                                FB_Bacnet.StartStopCommand_072.bEnWrite := TRUE;
                                FB_Bacnet.StartStopCommand_072.bVal := FALSE;
                            10: 
                                
                                FB_Bacnet.StartStopCommand_073.bEnWrite := TRUE;
                                FB_Bacnet.StartStopCommand_073.bVal := FALSE;
                            11: 
                                
                                FB_Bacnet.StartStopCommand_074.bEnWrite := TRUE;
                                FB_Bacnet.StartStopCommand_074.bVal := FALSE;
                            12: 
                                
                                FB_Bacnet.StartStopCommand_075.bEnWrite := TRUE;
                                FB_Bacnet.StartStopCommand_075.bVal := FALSE;
                            13: 
                                
                                FB_Bacnet.StartStopCommand_076.bEnWrite := TRUE;
                                FB_Bacnet.StartStopCommand_076.bVal := FALSE;
                            14: 
                                
                                FB_Bacnet.StartStopCommand_077.bEnWrite := TRUE;
                                FB_Bacnet.StartStopCommand_077.bVal := FALSE;
                            15: 
                                
                                FB_Bacnet.StartStopCommand_078.bEnWrite := TRUE;
                                FB_Bacnet.StartStopCommand_078.bVal := FALSE;
                            16: 
                                
                                FB_Bacnet.StartStopCommand_079.bEnWrite := TRUE;
                                FB_Bacnet.StartStopCommand_079.bVal := FALSE;
                            17: 
                                
                                FB_Bacnet.StartStopCommand_080.bEnWrite := TRUE;
                                FB_Bacnet.StartStopCommand_080.bVal := FALSE;
                            18: 
                                
                                FB_Bacnet.StartStopCommand_081.bEnWrite := TRUE;
                                FB_Bacnet.StartStopCommand_081.bVal := FALSE;
                            19: 
                                
                                FB_Bacnet.StartStopCommand_082.bEnWrite := TRUE;
                                FB_Bacnet.StartStopCommand_082.bVal := FALSE;
                            20: 
                                
                                FB_Bacnet.StartStopCommand_083.bEnWrite := TRUE;
                                FB_Bacnet.StartStopCommand_083.bVal := FALSE;
                            21: 
                                
                                FB_Bacnet.StartStopCommand_084.bEnWrite := TRUE;
                                FB_Bacnet.StartStopCommand_084.bVal := FALSE;
                            22: 
                                
                                FB_Bacnet.StartStopCommand_085.bEnWrite := TRUE;
                                FB_Bacnet.StartStopCommand_085.bVal := FALSE;
                            23: 
                                
                                FB_Bacnet.StartStopCommand_112.bEnWrite := TRUE;
                                FB_Bacnet.StartStopCommand_112.bVal := FALSE;
                            24: 
                                
                                FB_Bacnet.StartStopCommand_241.bEnWrite := TRUE;
                                FB_Bacnet.StartStopCommand_241.bVal := FALSE;
                            25: 
                                
                                FB_Bacnet.StartStopCommand_235.bEnWrite := TRUE;
                                FB_Bacnet.StartStopCommand_235.bVal := FALSE;
                        END_CASE
                    END_IF
                END_FOR
            END_IF
        END_IF
    END_IF
END_IF

END_FUNCTION_BLOCK

// ---- POUs/FB_Scheduler/FB_Scheduler_F52.TcPOU

      FUNCTION_BLOCK FB_Scheduler_F52
      VAR_INPUT
          currH : WORD;
          currM : WORD;
          currD : WORD;
      END_VAR
      VAR_IN_OUT
          FB_Bacnet : FB_BACnet_DAIKIN_MasterStation_III_No_10;
      END_VAR
      VAR
          i : INT;
          bUnitTriggered : BOOL := FALSE; // New flag to track execution
          prevMinute : WORD := 0;        // New variable to track the previous minute
      END_VAR
      VAR PERSISTENT
          //scheduler var
          bEnSchedF52_ : BOOL := FALSE;
          wSchedWDHourStartF52_ : WORD; 
          wSchedWDMinStartF52_ : WORD; 
          wSchedWEHourStartF52_ : WORD; 
          wSchedWEMinStartF52_ : WORD;
          wSchedWDHourEndF52_ : WORD;
          wSchedWDMinEndF52_ : WORD;
          wSchedWEHourEndF52_ : WORD;
          wSchedWEMinEndF52_ : WORD;
          //unit var
          bUnitF52_ : ARRAY [1..23] OF BOOL;
      END_VAR


        // Reset trigger flag at minute change or at the exact scheduled time
        IF currM <> prevMinute OR 
           (currH = wSchedWDHourStartF52_ AND currM = wSchedWDMinStartF52_) OR 
           (currH = wSchedWDHourEndF52_ AND currM = wSchedWDMinEndF52_) THEN
            bUnitTriggered := FALSE;
            prevMinute := currM;
        END_IF

        // Unit Schedule Enable
        IF bEnSchedF52_ THEN
            // Weekday schedule
            IF currD >= 1 AND currD <= 5 THEN
                IF (wSchedWDHourStartF52_ <> wSchedWDHourEndF52_ OR wSchedWDMinStartF52_ <> wSchedWDMinEndF52_) THEN
                    // Schedule Unit ON
                    IF wSchedWDHourStartF52_ = currH AND wSchedWDMinStartF52_ = currM AND NOT bUnitTriggered THEN
                        bUnitTriggered := TRUE;
                        FOR i := 1 TO 23 DO
                            //send command unit ON
                            IF bUnitF52_[i] = TRUE THEN 
                                CASE i OF
                                    1: 
                                        
                                        FB_Bacnet.StartStopCommand_128.bEnWrite := TRUE;
                                        FB_Bacnet.StartStopCommand_128.bVal := TRUE;
                                    2: 
                                        
                                        FB_Bacnet.StartStopCommand_129.bEnWrite := TRUE;
                                        FB_Bacnet.StartStopCommand_129.bVal := TRUE;
                                    3: 
                                        
                                        FB_Bacnet.StartStopCommand_130.bEnWrite := TRUE;
                                        FB_Bacnet.StartStopCommand_130.bVal := TRUE;
                                    4: 
                                        
                                        FB_Bacnet.StartStopCommand_131.bEnWrite := TRUE;
                                        FB_Bacnet.StartStopCommand_131.bVal := TRUE;
                                    5: 
                                        
                                        FB_Bacnet.StartStopCommand_132.bEnWrite := TRUE;
                                        FB_Bacnet.StartStopCommand_132.bVal := TRUE;
                                    6: 
                                        
                                        FB_Bacnet.StartStopCommand_133.bEnWrite := TRUE;
                                        FB_Bacnet.StartStopCommand_133.bVal := TRUE;
                                    7: 
                                        
                                        FB_Bacnet.StartStopCommand_134.bEnWrite := TRUE;
                                        FB_Bacnet.StartStopCommand_134.bVal := TRUE;
                                    8: 
                                        
                                        FB_Bacnet.StartStopCommand_135.bEnWrite := TRUE;
                                        FB_Bacnet.StartStopCommand_135.bVal := TRUE;
                                    9: 
                                        
                                        FB_Bacnet.StartStopCommand_136.bEnWrite := TRUE;
                                        FB_Bacnet.StartStopCommand_136.bVal := TRUE;
                                    10: 
                                        
                                        FB_Bacnet.StartStopCommand_137.bEnWrite := TRUE;
                                        FB_Bacnet.StartStopCommand_137.bVal := TRUE;
                                    11: 
                                        
                                        FB_Bacnet.StartStopCommand_138.bEnWrite := TRUE;
                                        FB_Bacnet.StartStopCommand_138.bVal := TRUE;
                                    12: 
                                        
                                        FB_Bacnet.StartStopCommand_139.bEnWrite := TRUE;
                                        FB_Bacnet.StartStopCommand_139.bVal := TRUE;
                                    13: 
                                        
                                        FB_Bacnet.StartStopCommand_140.bEnWrite := TRUE;
                                        FB_Bacnet.StartStopCommand_140.bVal := TRUE;
                                    14: 
                                        
                                        FB_Bacnet.StartStopCommand_141.bEnWrite := TRUE;
                                        FB_Bacnet.StartStopCommand_141.bVal := TRUE;
                                    15: 
                                        
                                        FB_Bacnet.StartStopCommand_142.bEnWrite := TRUE;
                                        FB_Bacnet.StartStopCommand_142.bVal := TRUE;
                                    16: 
                                        
                                        FB_Bacnet.StartStopCommand_143.bEnWrite := TRUE;
                                        FB_Bacnet.StartStopCommand_143.bVal := TRUE;
                                    17: 
                                        
                                        FB_Bacnet.StartStopCommand_144.bEnWrite := TRUE;
                                        FB_Bacnet.StartStopCommand_144.bVal := TRUE;
                                    18: 
                                        
                                        FB_Bacnet.StartStopCommand_145.bEnWrite := TRUE;
                                        FB_Bacnet.StartStopCommand_145.bVal := TRUE;
                                    19: 
                                        
                                        FB_Bacnet.StartStopCommand_146.bEnWrite := TRUE;
                                        FB_Bacnet.StartStopCommand_146.bVal := TRUE;
                                    20: 
                                        
                                        FB_Bacnet.StartStopCommand_147.bEnWrite := TRUE;
                                        FB_Bacnet.StartStopCommand_147.bVal := TRUE;
                                    21: 
                                        
                                        FB_Bacnet.StartStopCommand_148.bEnWrite := TRUE;
                                        FB_Bacnet.StartStopCommand_148.bVal := TRUE;
                                    22: 
                                        
                                        FB_Bacnet.StartStopCommand_149.bEnWrite := TRUE;
                                        FB_Bacnet.StartStopCommand_149.bVal := TRUE;
                                    23: 
                                        
                                        FB_Bacnet.StartStopCommand_236.bEnWrite := TRUE;
                                        FB_Bacnet.StartStopCommand_236.bVal := TRUE;
                                END_CASE
                            END_IF
                        END_FOR
                    END_IF
                    // Schedule Unit OFF
                    IF wSchedWDHourEndF52_ = currH AND wSchedWDMinEndF52_ = currM AND NOT bUnitTriggered THEN
                        bUnitTriggered := TRUE;
                        FOR i := 1 TO 23 DO
                            //send command unit OFF
                            IF bUnitF52_[i] = TRUE THEN 
                                CASE i OF
                                    1: 
                                        
                                        FB_Bacnet.StartStopCommand_128.bEnWrite := TRUE;
                                        FB_Bacnet.StartStopCommand_128.bVal := FALSE;
                                    2: 
                                        
                                        FB_Bacnet.StartStopCommand_129.bEnWrite := TRUE;
                                        FB_Bacnet.StartStopCommand_129.bVal := FALSE;
                                    3: 
                                        
                                        FB_Bacnet.StartStopCommand_130.bEnWrite := TRUE;
                                        FB_Bacnet.StartStopCommand_130.bVal := FALSE;
                                    4: 
                                        
                                        FB_Bacnet.StartStopCommand_131.bEnWrite := TRUE;
                                        FB_Bacnet.StartStopCommand_131.bVal := FALSE;
                                    5: 
                                        
                                        FB_Bacnet.StartStopCommand_132.bEnWrite := TRUE;
                                        FB_Bacnet.StartStopCommand_132.bVal := FALSE;
                                    6: 
                                        
                                        FB_Bacnet.StartStopCommand_133.bEnWrite := TRUE;
                                        FB_Bacnet.StartStopCommand_133.bVal := FALSE;
                                    7: 
                                        
                                        FB_Bacnet.StartStopCommand_134.bEnWrite := TRUE;
                                        FB_Bacnet.StartStopCommand_134.bVal := FALSE;
                                    8: 
                                        
                                        FB_Bacnet.StartStopCommand_135.bEnWrite := TRUE;
                                        FB_Bacnet.StartStopCommand_135.bVal := FALSE;
                                    9: 
                                        
                                        FB_Bacnet.StartStopCommand_136.bEnWrite := TRUE;
                                        FB_Bacnet.StartStopCommand_136.bVal := FALSE;
                                    10: 
                                        
                                        FB_Bacnet.StartStopCommand_137.bEnWrite := TRUE;
                                        FB_Bacnet.StartStopCommand_137.bVal := FALSE;
                                    11: 
                                        
                                        FB_Bacnet.StartStopCommand_138.bEnWrite := TRUE;
                                        FB_Bacnet.StartStopCommand_138.bVal := FALSE;
                                    12: 
                                        
                                        FB_Bacnet.StartStopCommand_139.bEnWrite := TRUE;
                                        FB_Bacnet.StartStopCommand_139.bVal := FALSE;
                                    13: 
                                        
                                        FB_Bacnet.StartStopCommand_140.bEnWrite := TRUE;
                                        FB_Bacnet.StartStopCommand_140.bVal := FALSE;
                                    14: 
                                        
                                        FB_Bacnet.StartStopCommand_141.bEnWrite := TRUE;
                                        FB_Bacnet.StartStopCommand_141.bVal := FALSE;
                                    15: 
                                        
                                        FB_Bacnet.StartStopCommand_142.bEnWrite := TRUE;
                                        FB_Bacnet.StartStopCommand_142.bVal := FALSE;
                                    16: 
                                        
                                        FB_Bacnet.StartStopCommand_143.bEnWrite := TRUE;
                                        FB_Bacnet.StartStopCommand_143.bVal := FALSE;
                                    17: 
                                        
                                        FB_Bacnet.StartStopCommand_144.bEnWrite := TRUE;
                                        FB_Bacnet.StartStopCommand_144.bVal := FALSE;
                                    18: 
                                        
                                        FB_Bacnet.StartStopCommand_145.bEnWrite := TRUE;
                                        FB_Bacnet.StartStopCommand_145.bVal := FALSE;
                                    19: 
                                        
                                        FB_Bacnet.StartStopCommand_146.bEnWrite := TRUE;
                                        FB_Bacnet.StartStopCommand_146.bVal := FALSE;
                                    20: 
                                        
                                        FB_Bacnet.StartStopCommand_147.bEnWrite := TRUE;
                                        FB_Bacnet.StartStopCommand_147.bVal := FALSE;
                                    21: 
                                        
                                        FB_Bacnet.StartStopCommand_148.bEnWrite := TRUE;
                                        FB_Bacnet.StartStopCommand_148.bVal := FALSE;
                                    22: 
                                        
                                        FB_Bacnet.StartStopCommand_149.bEnWrite := TRUE;
                                        FB_Bacnet.StartStopCommand_149.bVal := FALSE;
                                    23: 
                                        
                                        FB_Bacnet.StartStopCommand_236.bEnWrite := TRUE;
                                        FB_Bacnet.StartStopCommand_236.bVal := FALSE;
                                END_CASE
                            END_IF
                        END_FOR
                    END_IF
                END_IF
            END_IF

            // Weekend schedule
            IF currD = 0 OR currD = 6 THEN
                IF (wSchedWEHourStartF52_ <> wSchedWEHourEndF52_ OR wSchedWEMinStartF52_ <> wSchedWEMinEndF52_) THEN
                    // Schedule Unit ON
                    IF wSchedWEHourStartF52_ = currH AND wSchedWEMinStartF52_ = currM AND NOT bUnitTriggered THEN
                        bUnitTriggered := TRUE;
                        FOR i := 1 TO 23 DO
                            //send command unit ON
                            IF bUnitF52_[i] = TRUE THEN 
                                CASE i OF
                                    1: 
                                        
                                        FB_Bacnet.StartStopCommand_128.bEnWrite := TRUE;
                                        FB_Bacnet.StartStopCommand_128.bVal := TRUE;
                                    2: 
                                        
                                        FB_Bacnet.StartStopCommand_129.bEnWrite := TRUE;
                                        FB_Bacnet.StartStopCommand_129.bVal := TRUE;
                                    3: 
                                        
                                        FB_Bacnet.StartStopCommand_130.bEnWrite := TRUE;
                                        FB_Bacnet.StartStopCommand_130.bVal := TRUE;
                                    4: 
                                        
                                        FB_Bacnet.StartStopCommand_131.bEnWrite := TRUE;
                                        FB_Bacnet.StartStopCommand_131.bVal := TRUE;
                                    5: 
                                        
                                        FB_Bacnet.StartStopCommand_132.bEnWrite := TRUE;
                                        FB_Bacnet.StartStopCommand_132.bVal := TRUE;
                                    6: 
                                        
                                        FB_Bacnet.StartStopCommand_133.bEnWrite := TRUE;
                                        FB_Bacnet.StartStopCommand_133.bVal := TRUE;
                                    7: 
                                        
                                        FB_Bacnet.StartStopCommand_134.bEnWrite := TRUE;
                                        FB_Bacnet.StartStopCommand_134.bVal := TRUE;
                                    8: 
                                        
                                        FB_Bacnet.StartStopCommand_135.bEnWrite := TRUE;
                                        FB_Bacnet.StartStopCommand_135.bVal := TRUE;
                                    9: 
                                        
                                        FB_Bacnet.StartStopCommand_136.bEnWrite := TRUE;
                                        FB_Bacnet.StartStopCommand_136.bVal := TRUE;
                                    10: 
                                        
                                        FB_Bacnet.StartStopCommand_137.bEnWrite := TRUE;
                                        FB_Bacnet.StartStopCommand_137.bVal := TRUE;
                                    11: 
                                        
                                        FB_Bacnet.StartStopCommand_138.bEnWrite := TRUE;
                                        FB_Bacnet.StartStopCommand_138.bVal := TRUE;
                                    12: 
                                        
                                        FB_Bacnet.StartStopCommand_139.bEnWrite := TRUE;
                                        FB_Bacnet.StartStopCommand_139.bVal := TRUE;
                                    13: 
                                        
                                        FB_Bacnet.StartStopCommand_140.bEnWrite := TRUE;
                                        FB_Bacnet.StartStopCommand_140.bVal := TRUE;
                                    14: 
                                        
                                        FB_Bacnet.StartStopCommand_141.bEnWrite := TRUE;
                                        FB_Bacnet.StartStopCommand_141.bVal := TRUE;
                                    15: 
                                        
                                        FB_Bacnet.StartStopCommand_142.bEnWrite := TRUE;
                                        FB_Bacnet.StartStopCommand_142.bVal := TRUE;
                                    16: 
                                        
                                        FB_Bacnet.StartStopCommand_143.bEnWrite := TRUE;
                                        FB_Bacnet.StartStopCommand_143.bVal := TRUE;
                                    17: 
                                        
                                        FB_Bacnet.StartStopCommand_144.bEnWrite := TRUE;
                                        FB_Bacnet.StartStopCommand_144.bVal := TRUE;
                                    18: 
                                        
                                        FB_Bacnet.StartStopCommand_145.bEnWrite := TRUE;
                                        FB_Bacnet.StartStopCommand_145.bVal := TRUE;
                                    19: 
                                        
                                        FB_Bacnet.StartStopCommand_146.bEnWrite := TRUE;
                                        FB_Bacnet.StartStopCommand_146.bVal := TRUE;
                                    20: 
                                        
                                        FB_Bacnet.StartStopCommand_147.bEnWrite := TRUE;
                                        FB_Bacnet.StartStopCommand_147.bVal := TRUE;
                                    21: 
                                        
                                        FB_Bacnet.StartStopCommand_148.bEnWrite := TRUE;
                                        FB_Bacnet.StartStopCommand_148.bVal := TRUE;
                                    22: 
                                        
                                        FB_Bacnet.StartStopCommand_149.bEnWrite := TRUE;
                                        FB_Bacnet.StartStopCommand_149.bVal := TRUE;
                                    23: 
                                        
                                        FB_Bacnet.StartStopCommand_236.bEnWrite := TRUE;
                                        FB_Bacnet.StartStopCommand_236.bVal := TRUE;
                                END_CASE
                            END_IF
                        END_FOR
                    END_IF
                    // Schedule Unit OFF
                    IF wSchedWEHourEndF52_ = currH AND wSchedWEMinEndF52_ = currM AND NOT bUnitTriggered THEN
                        bUnitTriggered := TRUE;
                        FOR i := 1 TO 23 DO
                            //send command unit OFF
                            IF bUnitF52_[i] = TRUE THEN 
                                CASE i OF
                                    1: 
                                        
                                        FB_Bacnet.StartStopCommand_128.bEnWrite := TRUE;
                                        FB_Bacnet.StartStopCommand_128.bVal := FALSE;
                                    2: 
                                        
                                        FB_Bacnet.StartStopCommand_129.bEnWrite := TRUE;
                                        FB_Bacnet.StartStopCommand_129.bVal := FALSE;
                                    3: 
                                        
                                        FB_Bacnet.StartStopCommand_130.bEnWrite := TRUE;
                                        FB_Bacnet.StartStopCommand_130.bVal := FALSE;
                                    4: 
                                        
                                        FB_Bacnet.StartStopCommand_131.bEnWrite := TRUE;
                                        FB_Bacnet.StartStopCommand_131.bVal := FALSE;
                                    5: 
                                        
                                        FB_Bacnet.StartStopCommand_132.bEnWrite := TRUE;
                                        FB_Bacnet.StartStopCommand_132.bVal := FALSE;
                                    6: 
                                        
                                        FB_Bacnet.StartStopCommand_133.bEnWrite := TRUE;
                                        FB_Bacnet.StartStopCommand_133.bVal := FALSE;
                                    7: 
                                        
                                        FB_Bacnet.StartStopCommand_134.bEnWrite := TRUE;
                                        FB_Bacnet.StartStopCommand_134.bVal := FALSE;
                                    8: 
                                        
                                        FB_Bacnet.StartStopCommand_135.bEnWrite := TRUE;
                                        FB_Bacnet.StartStopCommand_135.bVal := FALSE;
                                    9: 
                                        
                                        FB_Bacnet.StartStopCommand_136.bEnWrite := TRUE;
                                        FB_Bacnet.StartStopCommand_136.bVal := FALSE;
                                    10: 
                                        
                                        FB_Bacnet.StartStopCommand_137.bEnWrite := TRUE;
                                        FB_Bacnet.StartStopCommand_137.bVal := FALSE;
                                    11: 
                                        
                                        FB_Bacnet.StartStopCommand_138.bEnWrite := TRUE;
                                        FB_Bacnet.StartStopCommand_138.bVal := FALSE;
                                    12: 
                                        
                                        FB_Bacnet.StartStopCommand_139.bEnWrite := TRUE;
                                        FB_Bacnet.StartStopCommand_139.bVal := FALSE;
                                    13: 
                                        
                                        FB_Bacnet.StartStopCommand_140.bEnWrite := TRUE;
                                        FB_Bacnet.StartStopCommand_140.bVal := FALSE;
                                    14: 
                                        
                                        FB_Bacnet.StartStopCommand_141.bEnWrite := TRUE;
                                        FB_Bacnet.StartStopCommand_141.bVal := FALSE;
                                    15: 
                                        
                                        FB_Bacnet.StartStopCommand_142.bEnWrite := TRUE;
                                        FB_Bacnet.StartStopCommand_142.bVal := FALSE;
                                    16: 
                                        
                                        FB_Bacnet.StartStopCommand_143.bEnWrite := TRUE;
                                        FB_Bacnet.StartStopCommand_143.bVal := FALSE;
                                    17: 
                                        
                                        FB_Bacnet.StartStopCommand_144.bEnWrite := TRUE;
                                        FB_Bacnet.StartStopCommand_144.bVal := FALSE;
                                    18: 
                                        
                                        FB_Bacnet.StartStopCommand_145.bEnWrite := TRUE;
                                        FB_Bacnet.StartStopCommand_145.bVal := FALSE;
                                    19: 
                                        
                                        FB_Bacnet.StartStopCommand_146.bEnWrite := TRUE;
                                        FB_Bacnet.StartStopCommand_146.bVal := FALSE;
                                    20: 
                                        
                                        FB_Bacnet.StartStopCommand_147.bEnWrite := TRUE;
                                        FB_Bacnet.StartStopCommand_147.bVal := FALSE;
                                    21: 
                                        
                                        FB_Bacnet.StartStopCommand_148.bEnWrite := TRUE;
                                        FB_Bacnet.StartStopCommand_148.bVal := FALSE;
                                    22: 
                                        
                                        FB_Bacnet.StartStopCommand_149.bEnWrite := TRUE;
                                        FB_Bacnet.StartStopCommand_149.bVal := FALSE;
                                    23: 
                                        
                                        FB_Bacnet.StartStopCommand_236.bEnWrite := TRUE;
                                        FB_Bacnet.StartStopCommand_236.bVal := FALSE;
                                END_CASE
                            END_IF
                        END_FOR
                    END_IF
                END_IF
            END_IF
        END_IF

END_FUNCTION_BLOCK

// ---- POUs/FB_Scheduler/FB_Scheduler_F53.TcPOU

    FUNCTION_BLOCK FB_Scheduler_F53
      VAR_INPUT
          currH : WORD;
          currM : WORD;
          currD : WORD;
      END_VAR
      VAR_IN_OUT
          FB_Bacnet : FB_BACnet_DAIKIN_MasterStation_III_No_10;
      END_VAR
      VAR
          i : INT;
          bUnitTriggered : BOOL := FALSE; // New flag to track execution
          prevMinute : WORD := 0;        // New variable to track the previous minute
      END_VAR
      VAR PERSISTENT
          //scheduler var
          bEnSchedF53_ : BOOL := FALSE;
          wSchedWDHourStartF53_ : WORD; 
          wSchedWDMinStartF53_ : WORD; 
          wSchedWEHourStartF53_ : WORD; 
          wSchedWEMinStartF53_ : WORD;
          wSchedWDHourEndF53_ : WORD;
          wSchedWDMinEndF53_ : WORD;
          wSchedWEHourEndF53_ : WORD;
          wSchedWEMinEndF53_ : WORD;
          //unit var
          bUnitF53_ : ARRAY [1..25] OF BOOL;
      END_VAR


// Reset trigger flag at minute change or at the exact scheduled time
IF currM <> prevMinute OR 
   (currH = wSchedWDHourStartF53_ AND currM = wSchedWDMinStartF53_) OR 
   (currH = wSchedWDHourEndF53_ AND currM = wSchedWDMinEndF53_) THEN
    bUnitTriggered := FALSE;
    prevMinute := currM;
END_IF

// Unit Schedule Enable
IF bEnSchedF53_ THEN
    // Weekday schedule
    IF currD >= 1 AND currD <= 5 THEN
        IF (wSchedWDHourStartF53_ <> wSchedWDHourEndF53_ OR wSchedWDMinStartF53_ <> wSchedWDMinEndF53_) THEN
            // Schedule Unit ON
            IF wSchedWDHourStartF53_ = currH AND wSchedWDMinStartF53_ = currM AND NOT bUnitTriggered THEN
                bUnitTriggered := TRUE;
                FOR i := 1 TO 25 DO
                    //send command unit ON
                    IF bUnitF53_[i] = TRUE THEN 
                        CASE i OF
                            1: 
                                FB_Bacnet.StartStopCommand_192.bEnWrite := TRUE;
                                FB_Bacnet.StartStopCommand_192.bVal := TRUE;
                            2: 
                                FB_Bacnet.StartStopCommand_193.bEnWrite := TRUE;
                                FB_Bacnet.StartStopCommand_193.bVal := TRUE;
                            3: 
                                FB_Bacnet.StartStopCommand_194.bEnWrite := TRUE;
                                FB_Bacnet.StartStopCommand_194.bVal := TRUE;
                            4: 
                                FB_Bacnet.StartStopCommand_195.bEnWrite := TRUE;
                                FB_Bacnet.StartStopCommand_195.bVal := TRUE;
                            5: 
                                FB_Bacnet.StartStopCommand_196.bEnWrite := TRUE;
                                FB_Bacnet.StartStopCommand_196.bVal := TRUE;
                            6: 
                                FB_Bacnet.StartStopCommand_197.bEnWrite := TRUE;
                                FB_Bacnet.StartStopCommand_197.bVal := TRUE;
                            7: 
                                FB_Bacnet.StartStopCommand_198.bEnWrite := TRUE;
                                FB_Bacnet.StartStopCommand_198.bVal := TRUE;
                            8: 
                                FB_Bacnet.StartStopCommand_199.bEnWrite := TRUE;
                                FB_Bacnet.StartStopCommand_199.bVal := TRUE;
                            9: 
                                //FB_Bacnet.StartStopCommand_200.bEnWrite := TRUE;
                                //FB_Bacnet.StartStopCommand_200.bVal := TRUE;
                            10: 
                                FB_Bacnet.StartStopCommand_201.bEnWrite := TRUE;
                                FB_Bacnet.StartStopCommand_201.bVal := TRUE;
                            11: 
                                FB_Bacnet.StartStopCommand_202.bEnWrite := TRUE;
                                FB_Bacnet.StartStopCommand_202.bVal := TRUE;
                            12: 
                                FB_Bacnet.StartStopCommand_203.bEnWrite := TRUE;
                                FB_Bacnet.StartStopCommand_203.bVal := TRUE;
                            13: 
                                FB_Bacnet.StartStopCommand_204.bEnWrite := TRUE;
                                FB_Bacnet.StartStopCommand_204.bVal := TRUE;
                            14: 
                                FB_Bacnet.StartStopCommand_205.bEnWrite := TRUE;
                                FB_Bacnet.StartStopCommand_205.bVal := TRUE;
                            15: 
                                FB_Bacnet.StartStopCommand_206.bEnWrite := TRUE;
                                FB_Bacnet.StartStopCommand_206.bVal := TRUE;
                            16: 
                                FB_Bacnet.StartStopCommand_207.bEnWrite := TRUE;
                                FB_Bacnet.StartStopCommand_207.bVal := TRUE;
                            17: 
                                FB_Bacnet.StartStopCommand_208.bEnWrite := TRUE;
                                FB_Bacnet.StartStopCommand_208.bVal := TRUE;
                            18: 
                                FB_Bacnet.StartStopCommand_209.bEnWrite := TRUE;
                                FB_Bacnet.StartStopCommand_209.bVal := TRUE;
                            19: 
                                FB_Bacnet.StartStopCommand_210.bEnWrite := TRUE;
                                FB_Bacnet.StartStopCommand_210.bVal := TRUE;
                            20: 
                                FB_Bacnet.StartStopCommand_211.bEnWrite := TRUE;
                                FB_Bacnet.StartStopCommand_211.bVal := TRUE;
                            21: 
                                FB_Bacnet.StartStopCommand_212.bEnWrite := TRUE;
                                FB_Bacnet.StartStopCommand_212.bVal := TRUE;
                            22: 
                                FB_Bacnet.StartStopCommand_213.bEnWrite := TRUE;
                                FB_Bacnet.StartStopCommand_213.bVal := TRUE;
                            23: 
                                FB_Bacnet.StartStopCommand_242.bEnWrite := TRUE;
                                FB_Bacnet.StartStopCommand_242.bVal := TRUE;
                            24: 
                                FB_Bacnet.StartStopCommand_243.bEnWrite := TRUE;
                                FB_Bacnet.StartStopCommand_243.bVal := TRUE;
                            25: 
                                FB_Bacnet.StartStopCommand_237.bEnWrite := TRUE;
                                FB_Bacnet.StartStopCommand_237.bVal := TRUE;
                        END_CASE
                    END_IF
                END_FOR
            END_IF
            // Schedule Unit OFF
            IF wSchedWDHourEndF53_ = currH AND wSchedWDMinEndF53_ = currM AND NOT bUnitTriggered THEN
                bUnitTriggered := TRUE;
                FOR i := 1 TO 25 DO
                    //send command unit OFF
                    IF bUnitF53_[i] = TRUE THEN 
                        CASE i OF
                            1: 
                                FB_Bacnet.StartStopCommand_192.bEnWrite := TRUE;
                                FB_Bacnet.StartStopCommand_192.bVal := FALSE;
                            2: 
                                FB_Bacnet.StartStopCommand_193.bEnWrite := TRUE;
                                FB_Bacnet.StartStopCommand_193.bVal := FALSE;
                            3: 
                                FB_Bacnet.StartStopCommand_194.bEnWrite := TRUE;
                                FB_Bacnet.StartStopCommand_194.bVal := FALSE;
                            4: 
                                FB_Bacnet.StartStopCommand_195.bEnWrite := TRUE;
                                FB_Bacnet.StartStopCommand_195.bVal := FALSE;
                            5: 
                                FB_Bacnet.StartStopCommand_196.bEnWrite := TRUE;
                                FB_Bacnet.StartStopCommand_196.bVal := FALSE;
                            6: 
                                FB_Bacnet.StartStopCommand_197.bEnWrite := TRUE;
                                FB_Bacnet.StartStopCommand_197.bVal := FALSE;
                            7: 
                                FB_Bacnet.StartStopCommand_198.bEnWrite := TRUE;
                                FB_Bacnet.StartStopCommand_198.bVal := FALSE;
                            8: 
                                FB_Bacnet.StartStopCommand_199.bEnWrite := TRUE;
                                FB_Bacnet.StartStopCommand_199.bVal := FALSE;
                            9: 
                                //FB_Bacnet.StartStopCommand_200.bEnWrite := TRUE;
                                //FB_Bacnet.StartStopCommand_200.bVal := FALSE;
                            10: 
                                FB_Bacnet.StartStopCommand_201.bEnWrite := TRUE;
                                FB_Bacnet.StartStopCommand_201.bVal := FALSE;
                            11: 
                                FB_Bacnet.StartStopCommand_202.bEnWrite := TRUE;
                                FB_Bacnet.StartStopCommand_202.bVal := FALSE;
                            12: 
                                FB_Bacnet.StartStopCommand_203.bEnWrite := TRUE;
                                FB_Bacnet.StartStopCommand_203.bVal := FALSE;
                            13: 
                                FB_Bacnet.StartStopCommand_204.bEnWrite := TRUE;
                                FB_Bacnet.StartStopCommand_204.bVal := FALSE;
                            14: 
                                FB_Bacnet.StartStopCommand_205.bEnWrite := TRUE;
                                FB_Bacnet.StartStopCommand_205.bVal := FALSE;
                            15: 
                                FB_Bacnet.StartStopCommand_206.bEnWrite := TRUE;
                                FB_Bacnet.StartStopCommand_206.bVal := FALSE;
                            16: 
                                FB_Bacnet.StartStopCommand_207.bEnWrite := TRUE;
                                FB_Bacnet.StartStopCommand_207.bVal := FALSE;
                            17: 
                                FB_Bacnet.StartStopCommand_208.bEnWrite := TRUE;
                                FB_Bacnet.StartStopCommand_208.bVal := FALSE;
                            18: 
                                FB_Bacnet.StartStopCommand_209.bEnWrite := TRUE;
                                FB_Bacnet.StartStopCommand_209.bVal := FALSE;
                            19: 
                                FB_Bacnet.StartStopCommand_210.bEnWrite := TRUE;
                                FB_Bacnet.StartStopCommand_210.bVal := FALSE;
                            20: 
                                FB_Bacnet.StartStopCommand_211.bEnWrite := TRUE;
                                FB_Bacnet.StartStopCommand_211.bVal := FALSE;
                            21: 
                                FB_Bacnet.StartStopCommand_212.bEnWrite := TRUE;
                                FB_Bacnet.StartStopCommand_212.bVal := FALSE;
                            22: 
                                FB_Bacnet.StartStopCommand_213.bEnWrite := TRUE;
                                FB_Bacnet.StartStopCommand_213.bVal := FALSE;
                            23: 
                                FB_Bacnet.StartStopCommand_242.bEnWrite := TRUE;
                                FB_Bacnet.StartStopCommand_242.bVal := FALSE;
                            24: 
                                FB_Bacnet.StartStopCommand_243.bEnWrite := TRUE;
                                FB_Bacnet.StartStopCommand_243.bVal := FALSE;
                            25: 
                                FB_Bacnet.StartStopCommand_237.bEnWrite := TRUE;
                                FB_Bacnet.StartStopCommand_237.bVal := FALSE;
                        END_CASE
                    END_IF
                END_FOR
            END_IF
        END_IF
    END_IF

    // Weekend schedule
    IF currD = 0 OR currD = 6 THEN
        IF (wSchedWEHourStartF53_ <> wSchedWEHourEndF53_ OR wSchedWEMinStartF53_ <> wSchedWEMinEndF53_) THEN
            // Schedule Unit ON
            IF wSchedWEHourStartF53_ = currH AND wSchedWEMinStartF53_ = currM AND NOT bUnitTriggered THEN
                bUnitTriggered := TRUE;
                FOR i := 1 TO 25 DO
                    //send command unit ON
                    IF bUnitF53_[i] = TRUE THEN 
                        CASE i OF
                            1: 
                                FB_Bacnet.StartStopCommand_192.bEnWrite := TRUE;
                                FB_Bacnet.StartStopCommand_192.bVal := TRUE;
                            2: 
                                FB_Bacnet.StartStopCommand_193.bEnWrite := TRUE;
                                FB_Bacnet.StartStopCommand_193.bVal := TRUE;
                            3: 
                                FB_Bacnet.StartStopCommand_194.bEnWrite := TRUE;
                                FB_Bacnet.StartStopCommand_194.bVal := TRUE;
                            4: 
                                FB_Bacnet.StartStopCommand_195.bEnWrite := TRUE;
                                FB_Bacnet.StartStopCommand_195.bVal := TRUE;
                            5: 
                                FB_Bacnet.StartStopCommand_196.bEnWrite := TRUE;
                                FB_Bacnet.StartStopCommand_196.bVal := TRUE;
                            6: 
                                FB_Bacnet.StartStopCommand_197.bEnWrite := TRUE;
                                FB_Bacnet.StartStopCommand_197.bVal := TRUE;
                            7: 
                                FB_Bacnet.StartStopCommand_198.bEnWrite := TRUE;
                                FB_Bacnet.StartStopCommand_198.bVal := TRUE;
                            8: 
                                FB_Bacnet.StartStopCommand_199.bEnWrite := TRUE;
                                FB_Bacnet.StartStopCommand_199.bVal := TRUE;
                            9: 
                                //FB_Bacnet.StartStopCommand_200.bEnWrite := TRUE;
                                //FB_Bacnet.StartStopCommand_200.bVal := TRUE;
                            10: 
                                FB_Bacnet.StartStopCommand_201.bEnWrite := TRUE;
                                FB_Bacnet.StartStopCommand_201.bVal := TRUE;
                            11: 
                                FB_Bacnet.StartStopCommand_202.bEnWrite := TRUE;
                                FB_Bacnet.StartStopCommand_202.bVal := TRUE;
                            12: 
                                FB_Bacnet.StartStopCommand_203.bEnWrite := TRUE;
                                FB_Bacnet.StartStopCommand_203.bVal := TRUE;
                            13: 
                                FB_Bacnet.StartStopCommand_204.bEnWrite := TRUE;
                                FB_Bacnet.StartStopCommand_204.bVal := TRUE;
                            14: 
                                FB_Bacnet.StartStopCommand_205.bEnWrite := TRUE;
                                FB_Bacnet.StartStopCommand_205.bVal := TRUE;
                            15: 
                                FB_Bacnet.StartStopCommand_206.bEnWrite := TRUE;
                                FB_Bacnet.StartStopCommand_206.bVal := TRUE;
                            16: 
                                FB_Bacnet.StartStopCommand_207.bEnWrite := TRUE;
                                FB_Bacnet.StartStopCommand_207.bVal := TRUE;
                            17: 
                                FB_Bacnet.StartStopCommand_208.bEnWrite := TRUE;
                                FB_Bacnet.StartStopCommand_208.bVal := TRUE;
                            18: 
                                FB_Bacnet.StartStopCommand_209.bEnWrite := TRUE;
                                FB_Bacnet.StartStopCommand_209.bVal := TRUE;
                            19: 
                                FB_Bacnet.StartStopCommand_210.bEnWrite := TRUE;
                                FB_Bacnet.StartStopCommand_210.bVal := TRUE;
                            20: 
                                FB_Bacnet.StartStopCommand_211.bEnWrite := TRUE;
                                FB_Bacnet.StartStopCommand_211.bVal := TRUE;
                            21: 
                                FB_Bacnet.StartStopCommand_212.bEnWrite := TRUE;
                                FB_Bacnet.StartStopCommand_212.bVal := TRUE;
                            22: 
                                FB_Bacnet.StartStopCommand_213.bEnWrite := TRUE;
                                FB_Bacnet.StartStopCommand_213.bVal := TRUE;
                            23: 
                                FB_Bacnet.StartStopCommand_242.bEnWrite := TRUE;
                                FB_Bacnet.StartStopCommand_242.bVal := TRUE;
                            24: 
                                FB_Bacnet.StartStopCommand_243.bEnWrite := TRUE;
                                FB_Bacnet.StartStopCommand_243.bVal := TRUE;
                            25: 
                                FB_Bacnet.StartStopCommand_237.bEnWrite := TRUE;
                                FB_Bacnet.StartStopCommand_237.bVal := TRUE;
                        END_CASE
                    END_IF
                END_FOR        
            END_IF
            // Schedule Unit OFF
            IF wSchedWEHourEndF53_ = currH AND wSchedWEMinEndF53_ = currM AND NOT bUnitTriggered THEN
                bUnitTriggered := TRUE;
                FOR i := 1 TO 25 DO
                    //send command unit OFF
                    IF bUnitF53_[i] = TRUE THEN 
                        CASE i OF
                            1: 
                                FB_Bacnet.StartStopCommand_192.bEnWrite := TRUE;
                                FB_Bacnet.StartStopCommand_192.bVal := FALSE;
                            2: 
                                FB_Bacnet.StartStopCommand_193.bEnWrite := TRUE;
                                FB_Bacnet.StartStopCommand_193.bVal := FALSE;
                            3: 
                                FB_Bacnet.StartStopCommand_194.bEnWrite := TRUE;
                                FB_Bacnet.StartStopCommand_194.bVal := FALSE;
                            4: 
                                FB_Bacnet.StartStopCommand_195.bEnWrite := TRUE;
                                FB_Bacnet.StartStopCommand_195.bVal := FALSE;
                            5: 
                                FB_Bacnet.StartStopCommand_196.bEnWrite := TRUE;
                                FB_Bacnet.StartStopCommand_196.bVal := FALSE;
                            6: 
                                FB_Bacnet.StartStopCommand_197.bEnWrite := TRUE;
                                FB_Bacnet.StartStopCommand_197.bVal := FALSE;
                            7: 
                                FB_Bacnet.StartStopCommand_198.bEnWrite := TRUE;
                                FB_Bacnet.StartStopCommand_198.bVal := FALSE;
                            8: 
                                FB_Bacnet.StartStopCommand_199.bEnWrite := TRUE;
                                FB_Bacnet.StartStopCommand_199.bVal := FALSE;
                            9: 
                                //FB_Bacnet.StartStopCommand_200.bEnWrite := TRUE;
                                //FB_Bacnet.StartStopCommand_200.bVal := FALSE;
                            10: 
                                FB_Bacnet.StartStopCommand_201.bEnWrite := TRUE;
                                FB_Bacnet.StartStopCommand_201.bVal := FALSE;
                            11: 
                                FB_Bacnet.StartStopCommand_202.bEnWrite := TRUE;
                                FB_Bacnet.StartStopCommand_202.bVal := FALSE;
                            12: 
                                FB_Bacnet.StartStopCommand_203.bEnWrite := TRUE;
                                FB_Bacnet.StartStopCommand_203.bVal := FALSE;
                            13: 
                                FB_Bacnet.StartStopCommand_204.bEnWrite := TRUE;
                                FB_Bacnet.StartStopCommand_204.bVal := FALSE;
                            14: 
                                FB_Bacnet.StartStopCommand_205.bEnWrite := TRUE;
                                FB_Bacnet.StartStopCommand_205.bVal := FALSE;
                            15: 
                                FB_Bacnet.StartStopCommand_206.bEnWrite := TRUE;
                                FB_Bacnet.StartStopCommand_206.bVal := FALSE;
                            16: 
                                FB_Bacnet.StartStopCommand_207.bEnWrite := TRUE;
                                FB_Bacnet.StartStopCommand_207.bVal := FALSE;
                            17: 
                                FB_Bacnet.StartStopCommand_208.bEnWrite := TRUE;
                                FB_Bacnet.StartStopCommand_208.bVal := FALSE;
                            18: 
                                FB_Bacnet.StartStopCommand_209.bEnWrite := TRUE;
                                FB_Bacnet.StartStopCommand_209.bVal := FALSE;
                            19: 
                                FB_Bacnet.StartStopCommand_210.bEnWrite := TRUE;
                                FB_Bacnet.StartStopCommand_210.bVal := FALSE;
                            20: 
                                FB_Bacnet.StartStopCommand_211.bEnWrite := TRUE;
                                FB_Bacnet.StartStopCommand_211.bVal := FALSE;
                            21: 
                                FB_Bacnet.StartStopCommand_212.bEnWrite := TRUE;
                                FB_Bacnet.StartStopCommand_212.bVal := FALSE;
                            22: 
                                FB_Bacnet.StartStopCommand_213.bEnWrite := TRUE;
                                FB_Bacnet.StartStopCommand_213.bVal := FALSE;
                            23: 
                                FB_Bacnet.StartStopCommand_242.bEnWrite := TRUE;
                                FB_Bacnet.StartStopCommand_242.bVal := FALSE;
                            24: 
                                FB_Bacnet.StartStopCommand_243.bEnWrite := TRUE;
                                FB_Bacnet.StartStopCommand_243.bVal := FALSE;
                            25: 
                                FB_Bacnet.StartStopCommand_237.bEnWrite := TRUE;
                                FB_Bacnet.StartStopCommand_237.bVal := FALSE;
                        END_CASE
                    END_IF
                END_FOR
            END_IF
        END_IF
    END_IF
END_IF

END_FUNCTION_BLOCK

// ---- POUs/FB_Scheduler/FB_Scheduler_F55.TcPOU

      FUNCTION_BLOCK FB_Scheduler_F55
      VAR_INPUT
          currH : WORD;
          currM : WORD;
          currD : WORD;
      END_VAR
      VAR_IN_OUT
          FB_Bacnet : FB_BACnet_DAIKIN_MasterStation_III_No_10;
      END_VAR
      VAR
          i : INT;
          bUnitTriggered : BOOL := FALSE; // New flag to track execution
          prevMinute : WORD := 0;        // New variable to track the previous minute
      END_VAR
      VAR PERSISTENT
          //scheduler var
          bEnSchedF55_ : BOOL := FALSE;
          wSchedWDHourStartF55_ : WORD; 
          wSchedWDMinStartF55_ : WORD; 
          wSchedWEHourStartF55_ : WORD; 
          wSchedWEMinStartF55_ : WORD;
          wSchedWDHourEndF55_ : WORD;
          wSchedWDMinEndF55_ : WORD;
          wSchedWEHourEndF55_ : WORD;
          wSchedWEMinEndF55_ : WORD;
          //unit var
          bUnitF55_ : ARRAY [1..21] OF BOOL;
      END_VAR


        // Reset trigger flag at minute change or at the exact scheduled time
        IF currM <> prevMinute OR 
           (currH = wSchedWDHourStartF55_ AND currM = wSchedWDMinStartF55_) OR 
           (currH = wSchedWDHourEndF55_ AND currM = wSchedWDMinEndF55_) THEN
            bUnitTriggered := FALSE;
            prevMinute := currM;
        END_IF

        // Unit Schedule Enable
        IF bEnSchedF55_ THEN
            // Weekday schedule
            IF currD >= 1 AND currD <= 5 THEN
                IF (wSchedWDHourStartF55_ <> wSchedWDHourEndF55_ OR wSchedWDMinStartF55_ <> wSchedWDMinEndF55_) THEN
                    // Schedule Unit ON
                    IF wSchedWDHourStartF55_ = currH AND wSchedWDMinStartF55_ = currM AND NOT bUnitTriggered THEN
                        bUnitTriggered := TRUE;
                        FOR i := 1 TO 21 DO
                            //send command unit ON
                            IF bUnitF55_[i] = TRUE THEN 
                                CASE i OF
                                    1: 
                                        
                                        FB_Bacnet.StartStopCommand_214.bEnWrite := TRUE;
                                        FB_Bacnet.StartStopCommand_214.bVal := TRUE;
                                    2: 
                                        
                                        FB_Bacnet.StartStopCommand_215.bEnWrite := TRUE;
                                        FB_Bacnet.StartStopCommand_215.bVal := TRUE;
                                    3: 
                                        
                                        FB_Bacnet.StartStopCommand_216.bEnWrite := TRUE;
                                        FB_Bacnet.StartStopCommand_216.bVal := TRUE;
                                    4: 
                                        
                                        FB_Bacnet.StartStopCommand_217.bEnWrite := TRUE;
                                        FB_Bacnet.StartStopCommand_217.bVal := TRUE;
                                    5: 
                                        
                                        FB_Bacnet.StartStopCommand_218.bEnWrite := TRUE;
                                        FB_Bacnet.StartStopCommand_218.bVal := TRUE;
                                    6: 
                                        
                                        FB_Bacnet.StartStopCommand_219.bEnWrite := TRUE;
                                        FB_Bacnet.StartStopCommand_219.bVal := TRUE;
                                    7: 
                                        
                                        FB_Bacnet.StartStopCommand_220.bEnWrite := TRUE;
                                        FB_Bacnet.StartStopCommand_220.bVal := TRUE;
                                    8: 
                                        
                                        FB_Bacnet.StartStopCommand_221.bEnWrite := TRUE;
                                        FB_Bacnet.StartStopCommand_221.bVal := TRUE;
                                    9: 
                                        
                                        FB_Bacnet.StartStopCommand_222.bEnWrite := TRUE;
                                        FB_Bacnet.StartStopCommand_222.bVal := TRUE;
                                    10: 
                                        
                                        FB_Bacnet.StartStopCommand_223.bEnWrite := TRUE;
                                        FB_Bacnet.StartStopCommand_223.bVal := TRUE;
                                    11: 
                                        
                                        FB_Bacnet.StartStopCommand_224.bEnWrite := TRUE;
                                        FB_Bacnet.StartStopCommand_224.bVal := TRUE;
                                    12: 
                                        
                                        FB_Bacnet.StartStopCommand_225.bEnWrite := TRUE;
                                        FB_Bacnet.StartStopCommand_225.bVal := TRUE;
                                    13: 
                                        
                                        FB_Bacnet.StartStopCommand_226.bEnWrite := TRUE;
                                        FB_Bacnet.StartStopCommand_226.bVal := TRUE;
                                    14: 
                                        
                                        FB_Bacnet.StartStopCommand_227.bEnWrite := TRUE;
                                        FB_Bacnet.StartStopCommand_227.bVal := TRUE;
                                    15: 
                                        
                                        FB_Bacnet.StartStopCommand_228.bEnWrite := TRUE;
                                        FB_Bacnet.StartStopCommand_228.bVal := TRUE;
                                    16: 
                                        
                                        FB_Bacnet.StartStopCommand_229.bEnWrite := TRUE;
                                        FB_Bacnet.StartStopCommand_229.bVal := TRUE;
                                    17: 
                                        
                                        FB_Bacnet.StartStopCommand_230.bEnWrite := TRUE;
                                        FB_Bacnet.StartStopCommand_230.bVal := TRUE;
                                    18: 
                                        
                                        FB_Bacnet.StartStopCommand_231.bEnWrite := TRUE;
                                        FB_Bacnet.StartStopCommand_231.bVal := TRUE;
                                    19: 
                                        
                                        FB_Bacnet.StartStopCommand_232.bEnWrite := TRUE;
                                        FB_Bacnet.StartStopCommand_232.bVal := TRUE;
                                    20: 
                                        
                                        FB_Bacnet.StartStopCommand_233.bEnWrite := TRUE;
                                        FB_Bacnet.StartStopCommand_233.bVal := TRUE;
                                    21: 
                                        
                                        FB_Bacnet.StartStopCommand_238.bEnWrite := TRUE;
                                        FB_Bacnet.StartStopCommand_238.bVal := TRUE;
                                END_CASE
                            END_IF
                        END_FOR
                    END_IF
                    // Schedule Unit OFF
                    IF wSchedWDHourEndF55_ = currH AND wSchedWDMinEndF55_ = currM AND NOT bUnitTriggered THEN
                        bUnitTriggered := TRUE;
                        FOR i := 1 TO 21 DO
                            //send command unit OFF
                            IF bUnitF55_[i] = TRUE THEN 
                                CASE i OF
                                    1: 
                                        
                                        FB_Bacnet.StartStopCommand_214.bEnWrite := TRUE;
                                        FB_Bacnet.StartStopCommand_214.bVal := FALSE;
                                    2: 
                                        
                                        FB_Bacnet.StartStopCommand_215.bEnWrite := TRUE;
                                        FB_Bacnet.StartStopCommand_215.bVal := FALSE;
                                    3: 
                                        
                                        FB_Bacnet.StartStopCommand_216.bEnWrite := TRUE;
                                        FB_Bacnet.StartStopCommand_216.bVal := FALSE;
                                    4: 
                                        
                                        FB_Bacnet.StartStopCommand_217.bEnWrite := TRUE;
                                        FB_Bacnet.StartStopCommand_217.bVal := FALSE;
                                    5: 
                                        
                                        FB_Bacnet.StartStopCommand_218.bEnWrite := TRUE;
                                        FB_Bacnet.StartStopCommand_218.bVal := FALSE;
                                    6: 
                                        
                                        FB_Bacnet.StartStopCommand_219.bEnWrite := TRUE;
                                        FB_Bacnet.StartStopCommand_219.bVal := FALSE;
                                    7: 
                                        
                                        FB_Bacnet.StartStopCommand_220.bEnWrite := TRUE;
                                        FB_Bacnet.StartStopCommand_220.bVal := FALSE;
                                    8: 
                                        
                                        FB_Bacnet.StartStopCommand_221.bEnWrite := TRUE;
                                        FB_Bacnet.StartStopCommand_221.bVal := FALSE;
                                    9: 
                                        
                                        FB_Bacnet.StartStopCommand_222.bEnWrite := TRUE;
                                        FB_Bacnet.StartStopCommand_222.bVal := FALSE;
                                    10: 
                                        
                                        FB_Bacnet.StartStopCommand_223.bEnWrite := TRUE;
                                        FB_Bacnet.StartStopCommand_223.bVal := FALSE;
                                    11: 
                                        
                                        FB_Bacnet.StartStopCommand_224.bEnWrite := TRUE;
                                        FB_Bacnet.StartStopCommand_224.bVal := FALSE;
                                    12: 
                                        
                                        FB_Bacnet.StartStopCommand_225.bEnWrite := TRUE;
                                        FB_Bacnet.StartStopCommand_225.bVal := FALSE;
                                    13: 
                                        
                                        FB_Bacnet.StartStopCommand_226.bEnWrite := TRUE;
                                        FB_Bacnet.StartStopCommand_226.bVal := FALSE;
                                    14: 
                                        
                                        FB_Bacnet.StartStopCommand_227.bEnWrite := TRUE;
                                        FB_Bacnet.StartStopCommand_227.bVal := FALSE;
                                    15: 
                                        
                                        FB_Bacnet.StartStopCommand_228.bEnWrite := TRUE;
                                        FB_Bacnet.StartStopCommand_228.bVal := FALSE;
                                    16: 
                                        
                                        FB_Bacnet.StartStopCommand_229.bEnWrite := TRUE;
                                        FB_Bacnet.StartStopCommand_229.bVal := FALSE;
                                    17: 
                                        
                                        FB_Bacnet.StartStopCommand_230.bEnWrite := TRUE;
                                        FB_Bacnet.StartStopCommand_230.bVal := FALSE;
                                    18: 
                                        
                                        FB_Bacnet.StartStopCommand_231.bEnWrite := TRUE;
                                        FB_Bacnet.StartStopCommand_231.bVal := FALSE;
                                    19: 
                                        
                                        FB_Bacnet.StartStopCommand_232.bEnWrite := TRUE;
                                        FB_Bacnet.StartStopCommand_232.bVal := FALSE;
                                    20: 
                                        
                                        FB_Bacnet.StartStopCommand_233.bEnWrite := TRUE;
                                        FB_Bacnet.StartStopCommand_233.bVal := FALSE;
                                    21: 
                                        
                                        FB_Bacnet.StartStopCommand_238.bEnWrite := TRUE;
                                        FB_Bacnet.StartStopCommand_238.bVal := FALSE;
                                END_CASE
                            END_IF
                        END_FOR
                    END_IF
                END_IF
            END_IF

            // Weekend schedule
            IF currD = 0 OR currD = 6 THEN
                IF (wSchedWEHourStartF55_ <> wSchedWEHourEndF55_ OR wSchedWEMinStartF55_ <> wSchedWEMinEndF55_) THEN
                    // Schedule Unit ON
                    IF wSchedWEHourStartF55_ = currH AND wSchedWEMinStartF55_ = currM AND NOT bUnitTriggered THEN
                        bUnitTriggered := TRUE;
                        FOR i := 1 TO 21 DO
                            //send command unit ON
                            IF bUnitF55_[i] = TRUE THEN 
                                CASE i OF
                                    1: 
                                        
                                        FB_Bacnet.StartStopCommand_214.bEnWrite := TRUE;
                                        FB_Bacnet.StartStopCommand_214.bVal := TRUE;
                                    2: 
                                        
                                        FB_Bacnet.StartStopCommand_215.bEnWrite := TRUE;
                                        FB_Bacnet.StartStopCommand_215.bVal := TRUE;
                                    3: 
                                        
                                        FB_Bacnet.StartStopCommand_216.bEnWrite := TRUE;
                                        FB_Bacnet.StartStopCommand_216.bVal := TRUE;
                                    4: 
                                        
                                        FB_Bacnet.StartStopCommand_217.bEnWrite := TRUE;
                                        FB_Bacnet.StartStopCommand_217.bVal := TRUE;
                                    5: 
                                        
                                        FB_Bacnet.StartStopCommand_218.bEnWrite := TRUE;
                                        FB_Bacnet.StartStopCommand_218.bVal := TRUE;
                                    6: 
                                        
                                        FB_Bacnet.StartStopCommand_219.bEnWrite := TRUE;
                                        FB_Bacnet.StartStopCommand_219.bVal := TRUE;
                                    7: 
                                        
                                        FB_Bacnet.StartStopCommand_220.bEnWrite := TRUE;
                                        FB_Bacnet.StartStopCommand_220.bVal := TRUE;
                                    8: 
                                        
                                        FB_Bacnet.StartStopCommand_221.bEnWrite := TRUE;
                                        FB_Bacnet.StartStopCommand_221.bVal := TRUE;
                                    9: 
                                        
                                        FB_Bacnet.StartStopCommand_222.bEnWrite := TRUE;
                                        FB_Bacnet.StartStopCommand_222.bVal := TRUE;
                                    10: 
                                        
                                        FB_Bacnet.StartStopCommand_223.bEnWrite := TRUE;
                                        FB_Bacnet.StartStopCommand_223.bVal := TRUE;
                                    11: 
                                        
                                        FB_Bacnet.StartStopCommand_224.bEnWrite := TRUE;
                                        FB_Bacnet.StartStopCommand_224.bVal := TRUE;
                                    12: 
                                        
                                        FB_Bacnet.StartStopCommand_225.bEnWrite := TRUE;
                                        FB_Bacnet.StartStopCommand_225.bVal := TRUE;
                                    13: 
                                        
                                        FB_Bacnet.StartStopCommand_226.bEnWrite := TRUE;
                                        FB_Bacnet.StartStopCommand_226.bVal := TRUE;
                                    14: 
                                        
                                        FB_Bacnet.StartStopCommand_227.bEnWrite := TRUE;
                                        FB_Bacnet.StartStopCommand_227.bVal := TRUE;
                                    15: 
                                        
                                        FB_Bacnet.StartStopCommand_228.bEnWrite := TRUE;
                                        FB_Bacnet.StartStopCommand_228.bVal := TRUE;
                                    16: 
                                        
                                        FB_Bacnet.StartStopCommand_229.bEnWrite := TRUE;
                                        FB_Bacnet.StartStopCommand_229.bVal := TRUE;
                                    17: 
                                        
                                        FB_Bacnet.StartStopCommand_230.bEnWrite := TRUE;
                                        FB_Bacnet.StartStopCommand_230.bVal := TRUE;
                                    18: 
                                        
                                        FB_Bacnet.StartStopCommand_231.bEnWrite := TRUE;
                                        FB_Bacnet.StartStopCommand_231.bVal := TRUE;
                                    19: 
                                        
                                        FB_Bacnet.StartStopCommand_232.bEnWrite := TRUE;
                                        FB_Bacnet.StartStopCommand_232.bVal := TRUE;
                                    20: 
                                        
                                        FB_Bacnet.StartStopCommand_233.bEnWrite := TRUE;
                                        FB_Bacnet.StartStopCommand_233.bVal := TRUE;
                                    21: 
                                        
                                        FB_Bacnet.StartStopCommand_238.bEnWrite := TRUE;
                                        FB_Bacnet.StartStopCommand_238.bVal := TRUE;
                                END_CASE
                            END_IF
                        END_FOR        
                    END_IF
                    // Schedule Unit OFF
                    IF wSchedWEHourEndF55_ = currH AND wSchedWEMinEndF55_ = currM AND NOT bUnitTriggered THEN
                        bUnitTriggered := TRUE;
                        FOR i := 1 TO 21 DO
                            //send command unit OFF
                            IF bUnitF55_[i] = TRUE THEN 
                                CASE i OF
                                    1: 
                                        
                                        FB_Bacnet.StartStopCommand_214.bEnWrite := TRUE;
                                        FB_Bacnet.StartStopCommand_214.bVal := FALSE;
                                    2: 
                                        
                                        FB_Bacnet.StartStopCommand_215.bEnWrite := TRUE;
                                        FB_Bacnet.StartStopCommand_215.bVal := FALSE;
                                    3: 
                                        
                                        FB_Bacnet.StartStopCommand_216.bEnWrite := TRUE;
                                        FB_Bacnet.StartStopCommand_216.bVal := FALSE;
                                    4: 
                                        
                                        FB_Bacnet.StartStopCommand_217.bEnWrite := TRUE;
                                        FB_Bacnet.StartStopCommand_217.bVal := FALSE;
                                    5: 
                                        
                                        FB_Bacnet.StartStopCommand_218.bEnWrite := TRUE;
                                        FB_Bacnet.StartStopCommand_218.bVal := FALSE;
                                    6: 
                                        
                                        FB_Bacnet.StartStopCommand_219.bEnWrite := TRUE;
                                        FB_Bacnet.StartStopCommand_219.bVal := FALSE;
                                    7: 
                                        
                                        FB_Bacnet.StartStopCommand_220.bEnWrite := TRUE;
                                        FB_Bacnet.StartStopCommand_220.bVal := FALSE;
                                    8: 
                                        
                                        FB_Bacnet.StartStopCommand_221.bEnWrite := TRUE;
                                        FB_Bacnet.StartStopCommand_221.bVal := FALSE;
                                    9: 
                                        
                                        FB_Bacnet.StartStopCommand_222.bEnWrite := TRUE;
                                        FB_Bacnet.StartStopCommand_222.bVal := FALSE;
                                    10: 
                                        
                                        FB_Bacnet.StartStopCommand_223.bEnWrite := TRUE;
                                        FB_Bacnet.StartStopCommand_223.bVal := FALSE;
                                    11: 
                                        
                                        FB_Bacnet.StartStopCommand_224.bEnWrite := TRUE;
                                        FB_Bacnet.StartStopCommand_224.bVal := FALSE;
                                    12: 
                                        
                                        FB_Bacnet.StartStopCommand_225.bEnWrite := TRUE;
                                        FB_Bacnet.StartStopCommand_225.bVal := FALSE;
                                    13: 
                                        
                                        FB_Bacnet.StartStopCommand_226.bEnWrite := TRUE;
                                        FB_Bacnet.StartStopCommand_226.bVal := FALSE;
                                    14: 
                                        
                                        FB_Bacnet.StartStopCommand_227.bEnWrite := TRUE;
                                        FB_Bacnet.StartStopCommand_227.bVal := FALSE;
                                    15: 
                                        
                                        FB_Bacnet.StartStopCommand_228.bEnWrite := TRUE;
                                        FB_Bacnet.StartStopCommand_228.bVal := FALSE;
                                    16: 
                                        
                                        FB_Bacnet.StartStopCommand_229.bEnWrite := TRUE;
                                        FB_Bacnet.StartStopCommand_229.bVal := FALSE;
                                    17: 
                                        
                                        FB_Bacnet.StartStopCommand_230.bEnWrite := TRUE;
                                        FB_Bacnet.StartStopCommand_230.bVal := FALSE;
                                    18: 
                                        
                                        FB_Bacnet.StartStopCommand_231.bEnWrite := TRUE;
                                        FB_Bacnet.StartStopCommand_231.bVal := FALSE;
                                    19: 
                                        
                                        FB_Bacnet.StartStopCommand_232.bEnWrite := TRUE;
                                        FB_Bacnet.StartStopCommand_232.bVal := FALSE;
                                    20: 
                                        
                                        FB_Bacnet.StartStopCommand_233.bEnWrite := TRUE;
                                        FB_Bacnet.StartStopCommand_233.bVal := FALSE;
                                    21: 
                                        
                                        FB_Bacnet.StartStopCommand_238.bEnWrite := TRUE;
                                        FB_Bacnet.StartStopCommand_238.bVal := FALSE;
                                END_CASE
                            END_IF
                        END_FOR
                    END_IF
                END_IF
            END_IF
        END_IF

END_FUNCTION_BLOCK

// ---- POUs/FB_Scheduler/FB_Scheduler_FPH1.TcPOU

      FUNCTION_BLOCK FB_Scheduler_FPH1
      VAR_INPUT
          currH : WORD;
          currM : WORD;
          currD : WORD;
      END_VAR
      VAR_IN_OUT
          FB_Bacnet : FB_BACnet_DAIKIN_MasterStation_III_No_10;
      END_VAR
      VAR
          i : INT;
          bUnitTriggered : BOOL := FALSE; // New flag to track execution
          prevMinute : WORD := 0;        // New variable to track the previous minute
      END_VAR
      VAR PERSISTENT
          //scheduler var
          bEnSchedFPH1_ : BOOL := FALSE;
          wSchedWDHourStartFPH1_ : WORD; 
          wSchedWDMinStartFPH1_ : WORD; 
          wSchedWEHourStartFPH1_ : WORD; 
          wSchedWEMinStartFPH1_ : WORD;
          wSchedWDHourEndFPH1_ : WORD;
          wSchedWDMinEndFPH1_ : WORD;
          wSchedWEHourEndFPH1_ : WORD;
          wSchedWEMinEndFPH1_ : WORD;
          //unit var
          bUnitFPH1_ : ARRAY [1..6] OF BOOL;
      END_VAR


        // Reset trigger flag at minute change or at the exact scheduled time
        IF currM <> prevMinute OR 
           (currH = wSchedWDHourStartFPH1_ AND currM = wSchedWDMinStartFPH1_) OR 
           (currH = wSchedWDHourEndFPH1_ AND currM = wSchedWDMinEndFPH1_) THEN
            bUnitTriggered := FALSE;
            prevMinute := currM;
        END_IF

        // Unit Schedule Enable
        IF bEnSchedFPH1_ THEN
            // Weekday schedule
            IF currD >= 1 AND currD <= 5 THEN
                IF (wSchedWDHourStartFPH1_ <> wSchedWDHourEndFPH1_ OR wSchedWDMinStartFPH1_ <> wSchedWDMinEndFPH1_) THEN
                    // Schedule Unit ON
                    IF wSchedWDHourStartFPH1_ = currH AND wSchedWDMinStartFPH1_ = currM AND NOT bUnitTriggered THEN
                        bUnitTriggered := TRUE;
                        FOR i := 1 TO 6 DO
                            // Send command unit ON
                            IF bUnitFPH1_[i] THEN 
                                CASE i OF
                                    1: FB_Bacnet.StartStopCommand_150.bEnWrite := TRUE;
                                       FB_Bacnet.StartStopCommand_150.bVal := TRUE;
                                    2: FB_Bacnet.StartStopCommand_151.bEnWrite := TRUE;
                                       FB_Bacnet.StartStopCommand_151.bVal := TRUE;
                                    3: 
                                        
                                        FB_Bacnet.StartStopCommand_152.bEnWrite := TRUE;
                                        FB_Bacnet.StartStopCommand_152.bVal := TRUE;
                                    4: 
                                        
                                        FB_Bacnet.StartStopCommand_153.bEnWrite := TRUE;
                                        FB_Bacnet.StartStopCommand_153.bVal := TRUE;
                                    5: 
                                        
                                        FB_Bacnet.StartStopCommand_154.bEnWrite := TRUE;
                                        FB_Bacnet.StartStopCommand_154.bVal := TRUE;
                                    6: 
                                        
                                        FB_Bacnet.StartStopCommand_155.bEnWrite := TRUE;
                                        FB_Bacnet.StartStopCommand_155.bVal := TRUE;
                                END_CASE
                            END_IF
                        END_FOR
                    END_IF
                    // Schedule Unit OFF
                    IF wSchedWDHourEndFPH1_ = currH AND wSchedWDMinEndFPH1_ = currM AND NOT bUnitTriggered THEN
                        bUnitTriggered := TRUE;
                        FOR i := 1 TO 6 DO
                            // Send command unit OFF
                            IF bUnitFPH1_[i] THEN 
                                CASE i OF
                                    1: FB_Bacnet.StartStopCommand_150.bEnWrite := TRUE;
                                       FB_Bacnet.StartStopCommand_150.bVal := FALSE;
                                    2: FB_Bacnet.StartStopCommand_151.bEnWrite := TRUE;
                                       FB_Bacnet.StartStopCommand_151.bVal := FALSE;
                                    3: 
                                        
                                        FB_Bacnet.StartStopCommand_152.bEnWrite := TRUE;
                                        FB_Bacnet.StartStopCommand_152.bVal := FALSE;
                                    4: 
                                        
                                        FB_Bacnet.StartStopCommand_153.bEnWrite := TRUE;
                                        FB_Bacnet.StartStopCommand_153.bVal := FALSE;
                                    5: 
                                        
                                        FB_Bacnet.StartStopCommand_154.bEnWrite := TRUE;
                                        FB_Bacnet.StartStopCommand_154.bVal := FALSE;
                                    6: 
                                        
                                        FB_Bacnet.StartStopCommand_155.bEnWrite := TRUE;
                                        FB_Bacnet.StartStopCommand_155.bVal := FALSE;
                                END_CASE
                            END_IF
                        END_FOR
                    END_IF
                END_IF
            END_IF
            // Weekend schedule
            IF currD = 0 OR currD = 6 THEN
                IF (wSchedWEHourStartFPH1_ <> wSchedWEHourEndFPH1_ OR wSchedWEMinStartFPH1_ <> wSchedWEMinEndFPH1_) THEN
                    // Schedule Unit ON
                    IF wSchedWEHourStartFPH1_ = currH AND wSchedWEMinStartFPH1_ = currM AND NOT bUnitTriggered THEN
                        bUnitTriggered := TRUE;
                        FOR i := 1 TO 6 DO
                            // Send command unit ON
                            IF bUnitFPH1_[i] THEN 
                                CASE i OF
                                    1: FB_Bacnet.StartStopCommand_150.bEnWrite := TRUE;
                                       FB_Bacnet.StartStopCommand_150.bVal := TRUE;
                                    2: FB_Bacnet.StartStopCommand_151.bEnWrite := TRUE;
                                       FB_Bacnet.StartStopCommand_151.bVal := TRUE;
                                    3: 
                                        
                                        FB_Bacnet.StartStopCommand_152.bEnWrite := TRUE;
                                        FB_Bacnet.StartStopCommand_152.bVal := TRUE;
                                    4: 
                                        
                                        FB_Bacnet.StartStopCommand_153.bEnWrite := TRUE;
                                        FB_Bacnet.StartStopCommand_153.bVal := TRUE;
                                    5: 
                                        
                                        FB_Bacnet.StartStopCommand_154.bEnWrite := TRUE;
                                        FB_Bacnet.StartStopCommand_154.bVal := TRUE;
                                    6: 
                                        
                                        FB_Bacnet.StartStopCommand_155.bEnWrite := TRUE;
                                        FB_Bacnet.StartStopCommand_155.bVal := TRUE;
                                END_CASE
                            END_IF
                        END_FOR
                    END_IF
                    // Schedule Unit OFF
                    IF wSchedWEHourEndFPH1_ = currH AND wSchedWEMinEndFPH1_ = currM AND NOT bUnitTriggered THEN
                        bUnitTriggered := TRUE;
                        FOR i := 1 TO 6 DO
                            // Send command unit OFF
                            IF bUnitFPH1_[i] THEN 
                                CASE i OF
                                    1: FB_Bacnet.StartStopCommand_150.bEnWrite := TRUE;
                                       FB_Bacnet.StartStopCommand_150.bVal := FALSE;
                                    2: FB_Bacnet.StartStopCommand_151.bEnWrite := TRUE;
                                       FB_Bacnet.StartStopCommand_151.bVal := FALSE;
                                    3: 
                                        
                                        FB_Bacnet.StartStopCommand_152.bEnWrite := TRUE;
                                        FB_Bacnet.StartStopCommand_152.bVal := FALSE;
                                    4: 
                                        
                                        FB_Bacnet.StartStopCommand_153.bEnWrite := TRUE;
                                        FB_Bacnet.StartStopCommand_153.bVal := FALSE;
                                    5: 
                                        
                                        FB_Bacnet.StartStopCommand_154.bEnWrite := TRUE;
                                        FB_Bacnet.StartStopCommand_154.bVal := FALSE;
                                    6: 
                                        
                                        FB_Bacnet.StartStopCommand_155.bEnWrite := TRUE;
                                        FB_Bacnet.StartStopCommand_155.bVal := FALSE;
                                END_CASE
                            END_IF
                        END_FOR
                    END_IF
                END_IF
            END_IF
        END_IF

END_FUNCTION_BLOCK

// ---- POUs/FB_Scheduler/FB_Scheduler_FPH2.TcPOU

      FUNCTION_BLOCK FB_Scheduler_FPH2
      VAR_INPUT
          currH : WORD;
          currM : WORD;
          currD : WORD;
      END_VAR
      VAR_IN_OUT
          FB_Bacnet : FB_BACnet_DAIKIN_MasterStation_III_No_10;
      END_VAR
      VAR
          i : INT;
          bUnitTriggered : BOOL := FALSE; // New flag to track execution
          prevMinute : WORD := 0;        // New variable to track the previous minute
      END_VAR
      VAR PERSISTENT
          //scheduler var
          bEnSchedFPH2_ : BOOL := FALSE;
          wSchedWDHourStartFPH2_ : WORD; 
          wSchedWDMinStartFPH2_ : WORD; 
          wSchedWEHourStartFPH2_ : WORD; 
          wSchedWEMinStartFPH2_ : WORD;
          wSchedWDHourEndFPH2_ : WORD;
          wSchedWDMinEndFPH2_ : WORD;
          wSchedWEHourEndFPH2_ : WORD;
          wSchedWEMinEndFPH2_ : WORD;
          //unit var
          bUnitFPH2_ : ARRAY [1..9] OF BOOL;
      END_VAR


        // Reset trigger flag at minute change or at the exact scheduled time
        IF currM <> prevMinute OR 
           (currH = wSchedWDHourStartFPH2_ AND currM = wSchedWDMinStartFPH2_) OR 
           (currH = wSchedWDHourEndFPH2_ AND currM = wSchedWDMinEndFPH2_) THEN
            bUnitTriggered := FALSE;
            prevMinute := currM;
        END_IF

        // Unit Schedule Enable
        IF bEnSchedFPH2_ THEN
            // Weekday schedule
            IF currD >= 1 AND currD <= 5 THEN
                IF (wSchedWDHourStartFPH2_ <> wSchedWDHourEndFPH2_ OR wSchedWDMinStartFPH2_ <> wSchedWDMinEndFPH2_) THEN
                    // Schedule Unit ON
                    IF wSchedWDHourStartFPH2_ = currH AND wSchedWDMinStartFPH2_ = currM AND NOT bUnitTriggered THEN
                        bUnitTriggered := TRUE;
                        FOR i := 1 TO 9 DO
                            // Send command unit ON
                            IF bUnitFPH2_[i] THEN 
                                CASE i OF
                                    1: FB_Bacnet.StartStopCommand_156.bEnWrite := TRUE;
                                       FB_Bacnet.StartStopCommand_156.bVal := TRUE;
                                    2: FB_Bacnet.StartStopCommand_157.bEnWrite := TRUE;
                                       FB_Bacnet.StartStopCommand_157.bVal := TRUE;
                                    3: FB_Bacnet.StartStopCommand_158.bEnWrite := TRUE;
                                       FB_Bacnet.StartStopCommand_158.bVal := TRUE;
                                    4: FB_Bacnet.StartStopCommand_159.bEnWrite := TRUE;
                                       FB_Bacnet.StartStopCommand_159.bVal := TRUE;
                                    5: FB_Bacnet.StartStopCommand_160.bEnWrite := TRUE;
                                       FB_Bacnet.StartStopCommand_160.bVal := TRUE;
                                    6: FB_Bacnet.StartStopCommand_161.bEnWrite := TRUE;
                                       FB_Bacnet.StartStopCommand_161.bVal := TRUE;
                                    7: FB_Bacnet.StartStopCommand_162.bEnWrite := TRUE;
                                       FB_Bacnet.StartStopCommand_162.bVal := TRUE;
                                    8: FB_Bacnet.StartStopCommand_163.bEnWrite := TRUE;
                                       FB_Bacnet.StartStopCommand_163.bVal := TRUE;
                                    9: FB_Bacnet.StartStopCommand_164.bEnWrite := TRUE;
                                       FB_Bacnet.StartStopCommand_164.bVal := TRUE;
                                END_CASE
                            END_IF
                        END_FOR
                    END_IF
                    // Schedule Unit OFF
                    IF wSchedWDHourEndFPH2_ = currH AND wSchedWDMinEndFPH2_ = currM AND NOT bUnitTriggered THEN
                        bUnitTriggered := TRUE;
                        FOR i := 1 TO 9 DO
                            // Send command unit OFF
                            IF bUnitFPH2_[i] THEN 
                                CASE i OF
                                    1: FB_Bacnet.StartStopCommand_156.bEnWrite := TRUE;
                                       FB_Bacnet.StartStopCommand_156.bVal := FALSE;
                                    2: FB_Bacnet.StartStopCommand_157.bEnWrite := TRUE;
                                       FB_Bacnet.StartStopCommand_157.bVal := FALSE;
                                    3: FB_Bacnet.StartStopCommand_158.bEnWrite := TRUE;
                                       FB_Bacnet.StartStopCommand_158.bVal := FALSE;
                                    4: FB_Bacnet.StartStopCommand_159.bEnWrite := TRUE;
                                       FB_Bacnet.StartStopCommand_159.bVal := FALSE;
                                    5: FB_Bacnet.StartStopCommand_160.bEnWrite := TRUE;
                                       FB_Bacnet.StartStopCommand_160.bVal := FALSE;
                                    6: FB_Bacnet.StartStopCommand_161.bEnWrite := TRUE;
                                       FB_Bacnet.StartStopCommand_161.bVal := FALSE;
                                    7: FB_Bacnet.StartStopCommand_162.bEnWrite := TRUE;
                                       FB_Bacnet.StartStopCommand_162.bVal := FALSE;
                                    8: FB_Bacnet.StartStopCommand_163.bEnWrite := TRUE;
                                       FB_Bacnet.StartStopCommand_163.bVal := FALSE;
                                    9: FB_Bacnet.StartStopCommand_164.bEnWrite := TRUE;
                                       FB_Bacnet.StartStopCommand_164.bVal := FALSE;
                                END_CASE
                            END_IF
                        END_FOR
                    END_IF
                END_IF
            END_IF
            // Weekend schedule
            IF currD = 0 OR currD = 6 THEN
                IF (wSchedWEHourStartFPH2_ <> wSchedWEHourEndFPH2_ OR wSchedWEMinStartFPH2_ <> wSchedWEMinEndFPH2_) THEN
                    // Schedule Unit ON
                    IF wSchedWEHourStartFPH2_ = currH AND wSchedWEMinStartFPH2_ = currM AND NOT bUnitTriggered THEN
                        bUnitTriggered := TRUE;
                        FOR i := 1 TO 9 DO
                            // Send command unit ON
                            IF bUnitFPH2_[i] THEN 
                                CASE i OF
                                    1: FB_Bacnet.StartStopCommand_156.bEnWrite := TRUE;
                                       FB_Bacnet.StartStopCommand_156.bVal := TRUE;
                                    2: FB_Bacnet.StartStopCommand_157.bEnWrite := TRUE;
                                       FB_Bacnet.StartStopCommand_157.bVal := TRUE;
                                    3: FB_Bacnet.StartStopCommand_158.bEnWrite := TRUE;
                                       FB_Bacnet.StartStopCommand_158.bVal := TRUE;
                                    4: FB_Bacnet.StartStopCommand_159.bEnWrite := TRUE;
                                       FB_Bacnet.StartStopCommand_159.bVal := TRUE;
                                    5: FB_Bacnet.StartStopCommand_160.bEnWrite := TRUE;
                                       FB_Bacnet.StartStopCommand_160.bVal := TRUE;
                                    6: FB_Bacnet.StartStopCommand_161.bEnWrite := TRUE;
                                       FB_Bacnet.StartStopCommand_161.bVal := TRUE;
                                    7: FB_Bacnet.StartStopCommand_162.bEnWrite := TRUE;
                                       FB_Bacnet.StartStopCommand_162.bVal := TRUE;
                                    8: FB_Bacnet.StartStopCommand_163.bEnWrite := TRUE;
                                       FB_Bacnet.StartStopCommand_163.bVal := TRUE;
                                    9: FB_Bacnet.StartStopCommand_164.bEnWrite := TRUE;
                                       FB_Bacnet.StartStopCommand_164.bVal := TRUE;
                                END_CASE
                            END_IF
                        END_FOR
                    END_IF
                    // Schedule Unit OFF
                    IF wSchedWEHourEndFPH2_ = currH AND wSchedWEMinEndFPH2_ = currM AND NOT bUnitTriggered THEN
                        bUnitTriggered := TRUE;
                        FOR i := 1 TO 9 DO
                            // Send command unit OFF
                            IF bUnitFPH2_[i] THEN 
                                CASE i OF
                                    1: FB_Bacnet.StartStopCommand_156.bEnWrite := TRUE;
                                       FB_Bacnet.StartStopCommand_156.bVal := FALSE;
                                    2: FB_Bacnet.StartStopCommand_157.bEnWrite := TRUE;
                                       FB_Bacnet.StartStopCommand_157.bVal := FALSE;
                                    3: FB_Bacnet.StartStopCommand_158.bEnWrite := TRUE;
                                       FB_Bacnet.StartStopCommand_158.bVal := FALSE;
                                    4: FB_Bacnet.StartStopCommand_159.bEnWrite := TRUE;
                                       FB_Bacnet.StartStopCommand_159.bVal := FALSE;
                                    5: FB_Bacnet.StartStopCommand_160.bEnWrite := TRUE;
                                       FB_Bacnet.StartStopCommand_160.bVal := FALSE;
                                    6: FB_Bacnet.StartStopCommand_161.bEnWrite := TRUE;
                                       FB_Bacnet.StartStopCommand_161.bVal := FALSE;
                                    7: FB_Bacnet.StartStopCommand_162.bEnWrite := TRUE;
                                       FB_Bacnet.StartStopCommand_162.bVal := FALSE;
                                    8: FB_Bacnet.StartStopCommand_163.bEnWrite := TRUE;
                                       FB_Bacnet.StartStopCommand_163.bVal := FALSE;
                                    9: FB_Bacnet.StartStopCommand_164.bEnWrite := TRUE;
                                       FB_Bacnet.StartStopCommand_164.bVal := FALSE;
                                END_CASE
                            END_IF
                        END_FOR
                    END_IF
                END_IF
            END_IF
        END_IF

END_FUNCTION_BLOCK

// ---- POUs/FB_Scheduler/FB_Scheduler_FPH3.TcPOU

